Yaskawa INFORM job: �k.JBI

/JOB
//NAME ‚k
//POS
///NPOS 4,0,0,0
///TOOL 0
///PULSE
C000=-12549,30472,-30846,8819,-163,8634
C001=-7029,38248,-27582,14195,3393,11126
C002=-30549,35416,-29406,14195,1965,9474
C003=-13413,41080,-20718,14027,3589,8466
//INST
///DATE 2014/09/13 22:43
///ATTR 0,0,0,0,0,0,0,0,0,0,0,0,0,1,0,0
///FRAME BASE
NOP
*‚k
MOVJ C000 VJ=100.00 CONT
MOVJ C001 VJ=100.00 CONT
MOVJ C002 VJ=60.00 CONT
MOVJ C003 VJ=100.00 CONT
JUMP *‚k
END
